FUNCTION TryConvert_BYTE_TO_DINT : BOOL
VAR_INPUT
	in : BYTE;
	out : REFERENCE TO DINT;
END_VAR

out := BYTE_TO_DINT(in);
TryConvert_BYTE_TO_DINT := TRUE;

END_FUNCTION

(* stored: Version 1.1.0.1, ProductVersion 3.1.4024.12
   POU TryConvert_BYTE_TO_DINT: Id {49294ad6-29aa-46c2-bbeb-526fcc020bbe}, SpecialFunc None *)
